Yaskawa INFORM job: MASTER_BATMAN_NEW_R1_NEW.JBI

/JOB
//NAME MASTER_BATMAN_NEW_R1_NEW
///FOLDERNAME SCIANA_WYPYCHAJACA_V19B_V20
//POS
///NPOS 7,7,7,0,0,0
///TOOL 0
///POSTYPE PULSE
///PULSE
C00000=5026,39564,34271,-3752,88090,85590
C00001=5026,39564,34271,-3752,88090,85590
C00002=5026,39564,34271,-3752,88090,52828
C00003=5643,128082,55348,12248,92639,-23986
C00004=7902,116420,10962,-11813,92779,-79531
C00005=29087,85831,-21148,-14422,96460,84613
C00006=5026,39564,34271,-3752,88090,-78121
BC00000=61339,583433,772029
BC00001=61339,583433,826968
BC00002=61339,583433,1035649
BC00003=65562,5048,1071913
BC00004=28128,212542,1075206
BC00005=125260,457132,1075157
BC00006=61339,583433,772029
EC00000=0,1
EC00001=-798157,-556476
EC00002=-798157,-556476
EC00003=-363194,-550745
EC00004=-798157,-556476
EC00005=-798157,-556476
EC00006=0,1
//INST
///DATE 2024/09/13 09:57
///ATTR SC,RW
///GROUP1 RB1,BS1
///GROUP2 ST1
NOP
MOVJ C00000 BC00000 VJ=100.00  +MOVJ EC00000 VJ=100.00
MOVJ C00001 BC00001 VJ=100.00  +MOVJ EC00001 VJ=100.00
PAUSE
PAUSE
'SCIAGNIJ USZY ZE SCIANY
MOVJ C00002 BC00002 VJ=100.00  +MOVJ EC00002 VJ=100.00
MOVJ C00003 BC00003 VJ=100.00  +MOVJ EC00003 VJ=100.00
COMM DOUT OT#(1433) ON
DOUT OT#(1435) ON
CALL JOB:BATMAN_ALL
MOVJ C00004 BC00004 VJ=50.00  +MOVJ EC00004 VJ=50.00
CALL JOB:BATMAN_2STR
MOVJ C00005 BC00005 VJ=50.00  +MOVJ EC00005 VJ=50.00
CALL JOB:BATMAN_4SPOINY
COMM DOUT OT#(1433) OFF
DOUT OT#(1435) OFF
MOVJ C00006 BC00006 VJ=100.00  +MOVJ EC00006 VJ=100.00
PAUSE
END
